SUBAPPLICATION mapping_Uebung_039 (* Spiegelabfolge V2 mit Schrittkette *)
  (* Standard: 61499-2 *)
  (* Version 1.0, 2023-10-23, franz *)
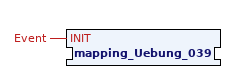
  EVENT_INPUT
    INIT;
  END_EVENT
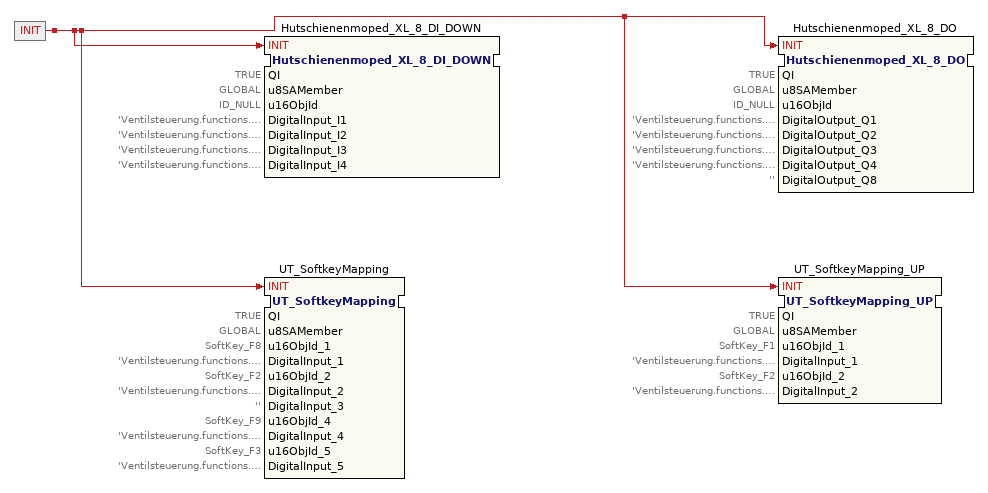
  FBS
    Hutschienenmoped_XL_8_DO : Hutschienenmoped_XL_8_DO(QI := TRUE, u8SAMember := GLOBAL, u16ObjId := ID_NULL, DigitalOutput_Q1 := 'Ventilsteuerung.functions.Q1.QX', DigitalOutput_Q2 := 'Ventilsteuerung.functions.Q2.QX', DigitalOutput_Q3 := 'Ventilsteuerung.functions.Q3.QX', DigitalOutput_Q4 := 'Ventilsteuerung.functions.Q4.QX', DigitalOutput_Q8 := '');
    UT_SoftkeyMapping_UP : UT_SoftkeyMapping_UP(QI := TRUE, u8SAMember := GLOBAL, u16ObjId_1 := SoftKey_F1, DigitalInput_1 := 'Ventilsteuerung.functions.SoftKey_F1_UP', u16ObjId_2 := SoftKey_F2, DigitalInput_2 := 'Ventilsteuerung.functions.SoftKey_F2_UP');
    Hutschienenmoped_XL_8_DI_DOWN : Hutschienenmoped_XL_8_DI_DOWN(QI := TRUE, u8SAMember := GLOBAL, u16ObjId := ID_NULL, DigitalInput_I1 := 'Ventilsteuerung.functions.DigitalInput_DOWN_I1', DigitalInput_I2 := 'Ventilsteuerung.functions.DigitalInput_DOWN_I2', DigitalInput_I3 := 'Ventilsteuerung.functions.DigitalInput_DOWN_I3', DigitalInput_I4 := 'Ventilsteuerung.functions.DigitalInput_DOWN_I4');
    UT_SoftkeyMapping : UT_SoftkeyMapping(QI := TRUE, u8SAMember := GLOBAL, u16ObjId_1 := SoftKey_F8, DigitalInput_1 := 'Ventilsteuerung.functions.Q1.IX', u16ObjId_2 := SoftKey_F2, DigitalInput_2 := 'Ventilsteuerung.functions.Q2.IX', DigitalInput_3 := '', u16ObjId_4 := SoftKey_F9, DigitalInput_4 := 'Ventilsteuerung.functions.Q3.IX', u16ObjId_5 := SoftKey_F3, DigitalInput_5 := 'Ventilsteuerung.functions.Q4.IX');
  END_FBS
  EVENT_CONNECTIONS
    INIT TO Hutschienenmoped_XL_8_DO.INIT;
    INIT TO UT_SoftkeyMapping_UP.INIT;
    INIT TO Hutschienenmoped_XL_8_DI_DOWN.INIT;
    INIT TO UT_SoftkeyMapping.INIT;
  END_CONNECTIONS
END_SUBAPPLICATION
